TYPE UDT_System_RD :
STRUCT
clock	: UDT_Clock_RD;
plcStatus :	UDT_PlcStatus_RD;				
programStatus	: UDT_ProgramStatus_RD;
 
END_STRUCT
END_TYPE

(* stored: Version 1.1.0.1, ProductVersion 3.1.4024.12
   DUT UDT_System_RD: Id {b47254ce-36f8-49c2-81c9-9623dcf823d3} *)
